// SIMATIC STEP 7 (V5.x) project TEMA 13 EJERCICIO 25
// CPU: CPU313 C-2 DP(1)
// station: P_ADR_BUS
// station: Hardware
// station: Equipo SIMATIC 300

DATA_BLOCK DB 1
VERSION : 0.1
  STRUCT
   M1 : BOOL ;
   M2 : BOOL ;
   M3 : BOOL ;
   M4 : BOOL ;
   M5 : BOOL ;
   M6 : BOOL ;
   M7 : BOOL ;
   M10 : BOOL ;
   M11 : BOOL ;
   M12 : BOOL ;
   M13 : BOOL ;
   M14 : BOOL ;
   M15 : BOOL ;
   M16 : BOOL ;
   M17 : BOOL ;
   M20 : BOOL ;
   M21 : BOOL ;
   M22 : BOOL ;
   M23 : BOOL ;
   M24 : BOOL ;
   M25 : BOOL ;
   M26 : BOOL ;
   M27 : BOOL ;
  END_STRUCT ;	
BEGIN
END_DATA_BLOCK

DATA_BLOCK DB 2
VERSION : 0.1
  STRUCT
   MARCA0 : BOOL ;
   MARCA1 : BOOL ;
   MARCA2 : BOOL ;
   MARCA3 : BOOL ;
   MARCA4 : BOOL ;
   MARCA5 : BOOL ;
   MARCA6 : BOOL ;
   MARCA7 : BOOL ;
   MARCA10 : BOOL ;
   MARCA11 : BOOL ;
   MARCA12 : BOOL ;
   MARCA13 : BOOL ;
   MARCA14 : BOOL ;
   MARCA15 : BOOL ;
   MARCA16 : BOOL ;
   MARCA17 : BOOL ;
  END_STRUCT ;	
BEGIN
END_DATA_BLOCK

DATA_BLOCK DB 3
VERSION : 0.1
  STRUCT
   MARCA0 : BOOL ;
   MARCA1 : BOOL ;
   MARCA2 : BOOL ;
   MARCA3 : BOOL ;
   MARCA4 : BOOL ;
   MARCA5 : BOOL ;
   MARCA6 : BOOL ;
   MARCA7 : BOOL ;
   MARCA10 : BOOL ;
   MARCA11 : BOOL ;
   MARCA12 : BOOL ;
   MARCA13 : BOOL ;
   MARCA14 : BOOL ;
   MARCA15 : BOOL ;
   MARCA16 : BOOL ;
   MARCA17 : BOOL ;
  END_STRUCT ;	
BEGIN
END_DATA_BLOCK

ORGANIZATION_BLOCK OB 1
TITLE = "Main Program Sweep (Cycle)"
//CLASIFICADOR AUTOMATICO DE CAJAS
VERSION : 0.1
VAR_TEMP
  OB1_EV_CLASS : BYTE ;	//Bits 0-3 = 1 (Coming event), Bits 4-7 = 1 (Event class 1)
  OB1_SCAN_1 : BYTE ;	//1 (Cold restart scan 1 of OB 1), 3 (Scan 2-n of OB 1)
  OB1_PRIORITY : BYTE ;	//Priority of OB Execution
  OB1_OB_NUMBR : BYTE ;	//1 (Organization block 1, OB1)
  OB1_RESERVED_1 : BYTE ;	//Reserved for system
  OB1_RESERVED_2 : BYTE ;	//Reserved for system
  OB1_PREV_CYCLE : INT ;	//Cycle time of previous OB1 scan (milliseconds)
  OB1_MIN_CYCLE : INT ;	//Minimum cycle time of OB1 (milliseconds)
  OB1_MAX_CYCLE : INT ;	//Maximum cycle time of OB1 (milliseconds)
  OB1_DATE_TIME : DATE_AND_TIME ;	//Date and time OB1 started
END_VAR
BEGIN
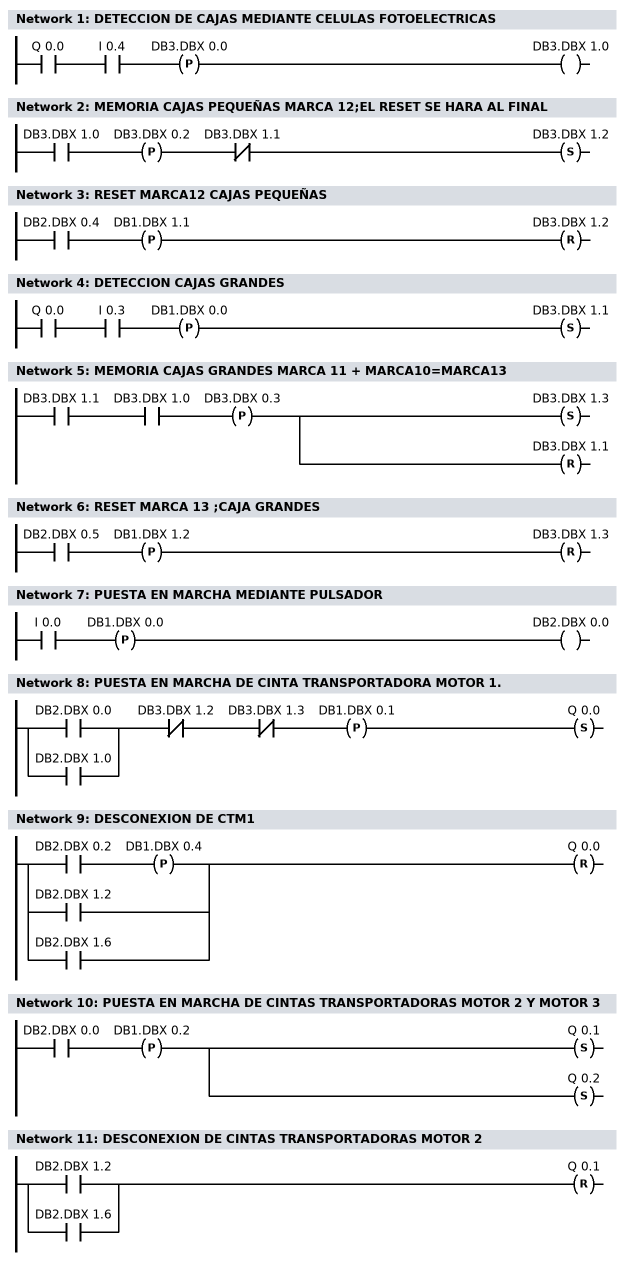
NETWORK
TITLE = DETECCION DE CAJAS MEDIANTE CELULAS FOTOELECTRICAS
//EXISTEN DOS TIPOS DE CAJAS PEQUEÑAS Y GRANDES.
//PARA RECONOCER LAS CAJAS PEQUEÑAS FCEL2 SE ACTIVARA YA QUE ESTA A LA ALTURA 
//OPORTUNA.
//PARA RECONOCER LAS CAJAS GRANDES SE TENDRA QUE ACTIVAR FCEL1 (NO PUEDE SER 
//ACTIVADO POR LAS CAJAS PEQUEÑAS POR QUE ESTA A LA ALTURA OPORTUNA)Y LUEGO FCEL2.
//ESTA INFORMACION SE TENDRA QUE GUARDAR EN UNA MEMORIA YA QUE EN CASO DE PARO,LA 
//MAQUINA UNA VEZ REANUDADA TENDRA QUE SEGUIR CON EL PROCESO CORRECTAMENTE.
//
//DETECCION CAJAS PEQUEÑAS
//
//
      A     Q 0.0;
      A     I 0.4;
      FP    DB3.DBX 0.0;
      =     DB3.DBX 1.0;
NETWORK
TITLE = MEMORIA CAJAS PEQUEÑAS MARCA 12;EL RESET SE HARA AL FINAL 
//COMO NECESITO QUE SE ACTIVE FCEL2 PARA REGISTRAR LA CAJAS GRANDES Y QUE NO ME 
//EJECUTE LA MEMORIA DE LAS PEQUEÑAS ,COLOCAREMOS OTRA MARCA AUXILIAR PARA QUE ME 
//PERMITA SUMAR LAS DOS SIN NECESIDAD DE CONFUNDIR A LA MAQUINA QUE SERA EN LA 
//CUAL INSERTE UN CONTACTO CERRADO PARA QUE SE HABRA UNA VEZ HALLA DETECTADO 
//FCEL1 Y ASI PODER UTILIZAR LA MARCA AUXILIAR.
      A     DB3.DBX 1.0;
      FP    DB3.DBX 0.2;
      AN    DB3.DBX 1.1;
      S     DB3.DBX 1.2;
NETWORK
TITLE = RESET MARCA12 CAJAS PEQUEÑAS
      A     DB2.DBX 0.4;
      FP    DB1.DBX 1.1;
      R     DB3.DBX 1.2;
NETWORK
TITLE = DETECCION CAJAS GRANDES
      A     Q 0.0;
      A     I 0.3;
      FP    DB1.DBX 0.0;
      S     DB3.DBX 1.1;
NETWORK
TITLE = MEMORIA CAJAS GRANDES MARCA 11 + MARCA10=MARCA13
//EL RESET DE LA MARCA SE HARA AL FINAL DEL PROCESO CUANDO YA NO SEA UTIL Y NOS 
//PERMITARA QUE LAS CELULAS FORTOELECTRICAS HAGAN SU FUNCION CORRECTAMENTE
      A     DB3.DBX 1.1;
      A     DB3.DBX 1.0;
      FP    DB3.DBX 0.3;
      S     DB3.DBX 1.3;
      R     DB3.DBX 1.1;
NETWORK
TITLE = RESET MARCA 13 ;CAJA GRANDES
      A     DB2.DBX 0.5;
      FP    DB1.DBX 1.2;
      R     DB3.DBX 1.3;
NETWORK
TITLE = PUESTA EN MARCHA MEDIANTE PULSADOR
//CUANDO PRESIONEMOS EL PULSADOR SE ACTIVARA EL PROCESO,ES DECIR,SE CONECTARAN 
//CTM1,CTM2,CTM3 Y LOS PISTONES ESTARAN PREPARADOS PARA CUANDO SEA NECESARIO
      A     I 0.0;
      FP    DB1.DBX 0.0;
      =     DB2.DBX 0.0;
NETWORK
TITLE = PUESTA EN MARCHA DE CINTA TRANSPORTADORA MOTOR 1.
//UN PULSO CONECTA CTM1 DE FORMA PERMANENTE
      A(;
      O     DB2.DBX 0.0;
      O     DB2.DBX 1.0;
      );
      AN    DB3.DBX 1.2;
      AN    DB3.DBX 1.3;
      FP    DB1.DBX 0.1;
      S     Q 0.0;
NETWORK
TITLE = DESCONEXION DE CTM1
//SE HARA EL RESET CUANDO CORRESPONDA:
//CUANDO LA CAJA PRESIONE EL F.C.FINAL LINEA.
//PARO.
//DESATIVACI0N.
      A     DB2.DBX 0.2;
      FP    DB1.DBX 0.4;
      O     DB2.DBX 1.2;
      O     DB2.DBX 1.6;
      R     Q 0.0;
NETWORK
TITLE = PUESTA EN MARCHA DE CINTAS TRANSPORTADORAS MOTOR 2 Y MOTOR 3 
//COMO ESTAS 2 CINTAS TRANSPORTADORAS FUNCIONAN  BAJO LAS MISMAS CONDIDICIONES 
//LOS 
//FACTORES QUE LAS CONECTAN Y DESCONECTAN SERAN LOS MISMOS.
      A     DB2.DBX 0.0;
      FP    DB1.DBX 0.2;
      S     Q 0.1;
      S     Q 0.2;
NETWORK
TITLE = DESCONEXION DE CINTAS TRANSPORTADORAS MOTOR 2  
//SE HARA EL RESET CUANDO CORRESPONDA:
//PARO.
//DESACTIVACION.
      O     DB2.DBX 1.2;
      O     DB2.DBX 1.6;
      R     Q 0.1;
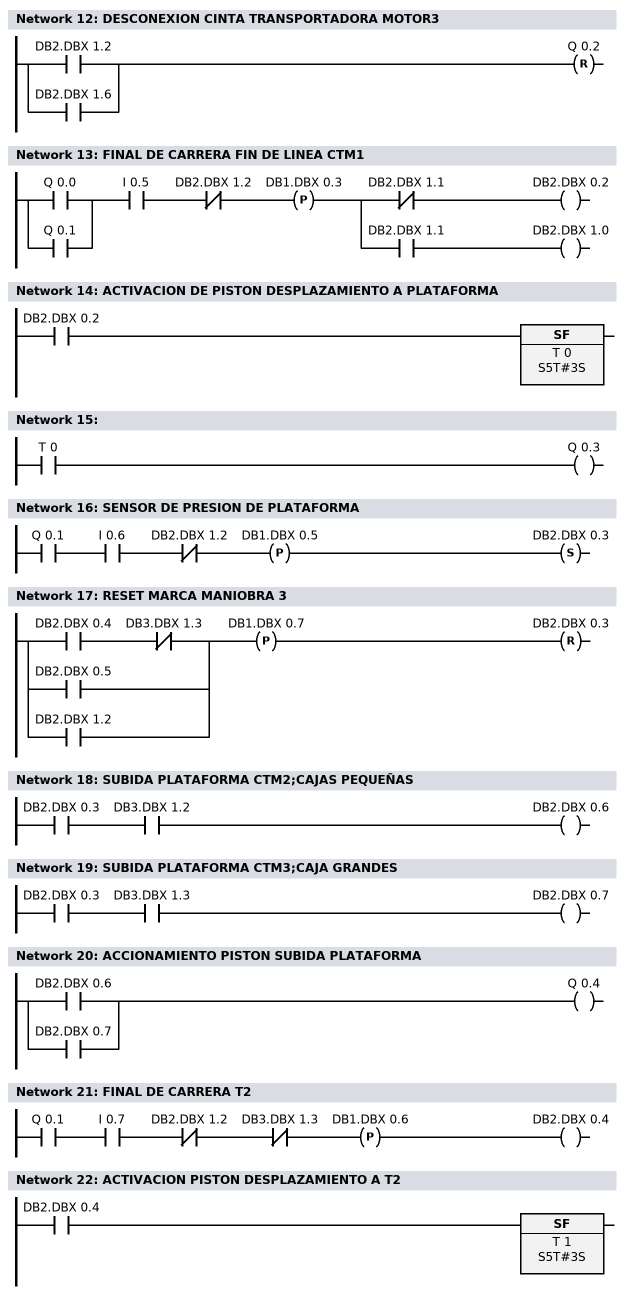
NETWORK
TITLE = DESCONEXION CINTA TRANSPORTADORA MOTOR3
//SE HARA EL RESET CUANDO CORRESPONDA:
//PARO.
//DESACTIVACION.
      O     DB2.DBX 1.2;
      O     DB2.DBX 1.6;
      R     Q 0.2;
NETWORK
TITLE = FINAL DE CARRERA FIN DE LINEA CTM1
//CUNADO UNA CAJA ACCIONE ESTE F.C. LA CTM1 SE PARARA Y ACTO SEGUIDO SE ACTIVARA 
//UN PISTON QUE DESPLAZARA LA CAJA SOBRE LA PLATAFORMA.
      A(;
      O     Q 0.0;
      O     Q 0.1;
      );
      A     I 0.5;
      AN    DB2.DBX 1.2;
      FP    DB1.DBX 0.3;
      =     L 20.0;
      A     L 20.0;
      AN    DB2.DBX 1.1;
      =     DB2.DBX 0.2;
      A     L 20.0;
      A     DB2.DBX 1.1;
      =     DB2.DBX 1.0;
NETWORK
TITLE = ACTIVACION DE PISTON DESPLAZAMIENTO A PLATAFORMA
//PARA SIMULAR EL ACCIONAMIENTO DE UN PISTON UTILIZO UN TEMPORIZADOR A LA 
//DESCONEXION QUE ALIMENTE UNA BOBINA(QUE ES EL PISTON) DURANTE 3 SEG.ES EL 
//TIEMPO 
//QUE TARDA EN DESPLAZARSE POR COMPLETO Y CUANDO SE APAGUE SE PRODUCIRA EL 
//RETORNO 
//POR RESORTE
      A     DB2.DBX 0.2;
      L     S5T#3S;
      SF    T 0;
NETWORK
TITLE =
      A     T 0;
      =     Q 0.3;
NETWORK
TITLE = SENSOR DE PRESION DE PLATAFORMA 
//UNA VEZ QUE EL SENSOR DE PRESION DETECTA UN PESO (EN ESTE CASO SERA CALIBRADO 
//PARA QUE CUALQUIERA DE LOS DOS TIPOS DE CAJAS LO ACTIVE) LA PLATAFORMA DEBERA 
//SUBIR A LA CINTA TRANSPORTADOA CORRESPODIENTE MEDIANTE UN PISTON 
      A     Q 0.1;
      A     I 0.6;
      AN    DB2.DBX 1.2;
      FP    DB1.DBX 0.5;
      S     DB2.DBX 0.3;
NETWORK
TITLE = RESET MARCA MANIOBRA 3
      A(;
      A     DB2.DBX 0.4;
      AN    DB3.DBX 1.3;
      O     DB2.DBX 0.5;
      O     DB2.DBX 1.2;
      );
      FP    DB1.DBX 0.7;
      R     DB2.DBX 0.3;
NETWORK
TITLE = SUBIDA PLATAFORMA CTM2;CAJAS PEQUEÑAS
//LA MARCA 12 ES LA QUE INDICA A LA PLATAFORMA DONDE TIENE QUE SUBIR Y SERA 
//INTERRUMPIDA POR SU FINAL DE CARRERA.CUANDO LAS MEMORIAS DE LAS CAJAS CAREZCAN 
//DE IMPORTANCIA SE HARA UN RESET
      A     DB2.DBX 0.3;
      A     DB3.DBX 1.2;
      =     DB2.DBX 0.6;
NETWORK
TITLE = SUBIDA PLATAFORMA CTM3;CAJA GRANDES
// LA MARCA 13 SE COMPORTA DE LA MISMA FORMA PERO SUBE HASTA CTM3
      A     DB2.DBX 0.3;
      A     DB3.DBX 1.3;
      =     DB2.DBX 0.7;
NETWORK
TITLE = ACCIONAMIENTO PISTON SUBIDA PLATAFORMA
      O     DB2.DBX 0.6;
      O     DB2.DBX 0.7;
      =     Q 0.4;
NETWORK
TITLE = FINAL DE CARRERA T2
//CUANDO SE ACCIONE SE PARARA LA SUBIDA DE LA PLATAFORMA E INICIARA SU RETROCESO 
//POR RESORTE,ACTIVARA EL PISTON DE DESPLAZAMIENTO A T2 Y HARA UN RESET DE LAS 
//MARCAS QUE YA NO SEAN UTILES PARA EL CORRECTO FUNCIONAMIENTO DEL PROCESO Y POR 
//LO TANTO ESTARAN PREPARADAS PARA LA SIGUIENTE SECUENCIA
      A     Q 0.1;
      A     I 0.7;
      AN    DB2.DBX 1.2;
      AN    DB3.DBX 1.3;
      FP    DB1.DBX 0.6;
      =     DB2.DBX 0.4;
NETWORK
TITLE = ACTIVACION PISTON DESPLAZAMIENTO A T2
//PARA SIMULAR EL PISTON UTILIZARE EL SISTEMA ANTERIOMENTE MENCIONADO
      A     DB2.DBX 0.4;
      L     S5T#3S;
      SF    T 1;
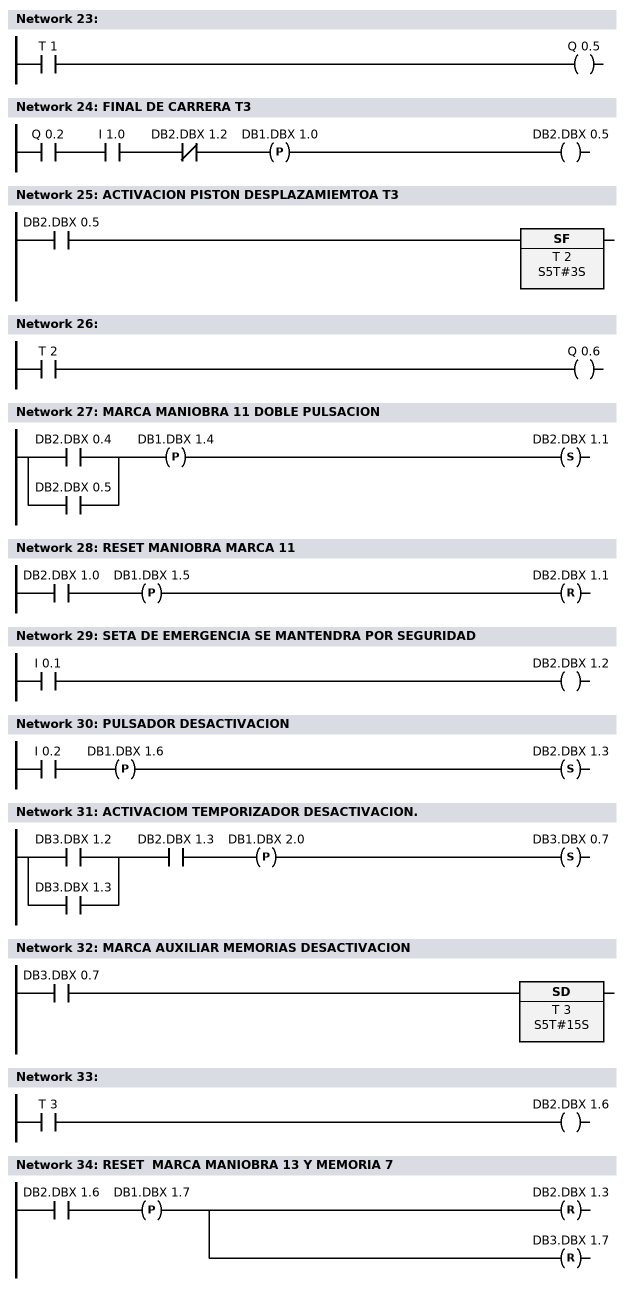
NETWORK
TITLE =
      A     T 1;
      =     Q 0.5;
NETWORK
TITLE = FINAL DE CARRERA T3
//EL SISTEMA SERA EL MISMO QUE EL ANTERIOMENTE CITADO
      A     Q 0.2;
      A     I 1.0;
      AN    DB2.DBX 1.2;
      FP    DB1.DBX 1.0;
      =     DB2.DBX 0.5;
NETWORK
TITLE = ACTIVACION PISTON DESPLAZAMIEMTOA T3
      A     DB2.DBX 0.5;
      L     S5T#3S;
      SF    T 2;
NETWORK
TITLE =
      A     T 2;
      =     Q 0.6;
NETWORK
TITLE = MARCA MANIOBRA 11 DOBLE PULSACION  
//CUANDO LA PLATAFORMA BAJE PRESIONARA OTRA VEZ EL F.C DE PLATAFORMA Y EN VEZ DE 
//PARAR CTM1 Y ACTIVAR PISTON DESPLAZAMIENTO SOLAMENTE ACTIVARA CTM1 Y LA 
//SIGUIENTE PULSACION PARARA CTM1 Y ACTIVARA PISTON. SE REPETIRA DE FORMA 
//INDEFINIDA.
      A(;
      O     DB2.DBX 0.4;
      O     DB2.DBX 0.5;
      );
      FP    DB1.DBX 1.4;
      S     DB2.DBX 1.1;
NETWORK
TITLE = RESET MANIOBRA MARCA 11
//SE HARA EL RESET CUANDO YA NO SEA NECESARIA,ES DECIR CUANDO ENTRE OTRA VEZ CTM1
      A     DB2.DBX 1.0;
      FP    DB1.DBX 1.5;
      R     DB2.DBX 1.1;
NETWORK
TITLE = SETA DE EMERGENCIA SE MANTENDRA POR SEGURIDAD
//AL PULSAR SE PARARA EL SISTEMA POR COMPLETO (LAS MEMORIAS DE MARCAS DE REGISTRO 
//DE CAJAS PERMANECERAN ACTIVAS PARA CUANDO SE ACTIVE EL SISTEMA DE NUEVO LA 
//MAQUINA SEPA DONDE SE ENCUENTRA Y ACTUE EN CONSECUENCIA) Y SE 
//CONDENARAN TODOS LOS FINALES DE CARRERA PARA EVITAR ACCIDENTES MIENTRAS SE 
//MANIPULE LA MAQUINA.
//MIENTRAS ESTE PRESIONADA LA SETA(RESET ALIMENTADO DE FORMA PERMANENTE) SERA 
//IMPOSIBLE HACER UN 
//SET EN LAS SALIDAS YA QUE PUEDE HABER RIESGO DE ACIONAMIENTO INVOLUNTARIO Y POR 
//LO TANTO UN FALLO FATAL.
//CONDICIONES DE PARO;
//PARO-LAS CINTAS ESTAN FUNCIONANDO,ES IRRELEVANTE.REINICIO NORMAL.
//PARO-FCEL1 DETECTA CAJA,ES IRRELEVANTE,LA MEMORIA PERMANECE REINICIO.NORMAL.
//PARO-FCEL2 DETECTA CAJA,ES IRRELEVANTE,LA MEMORIA PERMANECE REINICIO.NORMAL.
//PARO-CAJA PRESIONA F.C.F LINEA ,EL SIGUIENTE PASO SERIA DESCONECTAR CTM1 Y 
//ACTIVAR EL PISTON DE DESPLAZAMIENTO A PLATAFORMA UNA VEZ QUE HALLA DETECTADO 
//FCEL2 LA CAJA YA SE ENCUENTRA EN LA ZONA DE DESPLAZAMIENTO AL REINICIAR LA 
//MAQUINA ,EL F.C F LINEA ESTA PRESIONADO ASI QUE CTM1 NO FUNCIONA Y EL PISTON SE 
//DESPLAZA COLOCANDO LA CAJA EN LA PLATAFORMA.
//PARO-CAJA EN PLATAFORMA,EN ESTE CASO LAS MARCAS DE MEMORIA LAS QUE 
//INDIQUEN A LA MAQUINA DONDE SE ENCUENTRA Y DONDE DEBE DE IR(SI LA 
//PLATAFORMA ESTA SUBIENDO BAJARA A SU POSICION DE REPOSO).MARCHA CTM1 NO 
//FUNCIONA Y CTM2 Y CTM3 SI ,AL ESTAR PRESIONADO EL SENSOR DE PRESION LA 
//PLATAFORMA SUBIRA GOBERNADO POR LAS MARCAS DE MEMORIA DONDE CORRESPONDA.
      A     I 0.1;
      =     DB2.DBX 1.2;
NETWORK
TITLE = PULSADOR DESACTIVACION
//CON ESTE PULSADOR LO QUE CONSEGUINOS ES QUE EL SISTEMA DE FORMA INTELIGENTE 
//PARE 
//LA MAQUINA PERO NO AL INSTANTE ,EN EL CASO DE QUE HALLA INICIADO EL PROCESO(QUE 
//LAS CELULAS FOTOELECTRICAS HALLAN DETECTADO CAJA) DEJARA CONTINUAR HASTA 
//QUE TERMINE DE CLASIFICARLA Y NO PERMITIENDO QUE CIRCULE OTRA Y POR LO TANTO 
//ENTRA EN ESTADO DE REPOSO.CUANDO NO HALLA DETECTADO CAJA SE ACTIVARA LA 
//DESACTIVACION UNA VEZ ESTEN ACTIVAS LAS MARCAS DE MEMORIA 12 O 13.EL TIEMPO 
//ESTIMADO EN CLASIFICAR UNA CAJA DESDE QUE LAS CELULAS RECONOCEN CAJA HASTA QUE 
//LLEGAN A SU DESTINO ES DE 10 SEG.
//
      A     I 0.2;
      FP    DB1.DBX 1.6;
      S     DB2.DBX 1.3;
NETWORK
TITLE = ACTIVACIOM TEMPORIZADOR DESACTIVACION.
//PARA ACTUAR SOBRE ESTE TEMPORIZADOR UNA DE LAS MARCAS DE MEMORIA 12 O 13 TENDRAN
// 
//QUE ESTAR EN ON Y SI NO ES EL CASO ACTUARA CUANDO LO ESTE UNA DE LAS DOS.
      A(;
      O     DB3.DBX 1.2;
      O     DB3.DBX 1.3;
      );
      A     DB2.DBX 1.3;
      FP    DB1.DBX 2.0;
      S     DB3.DBX 0.7;
NETWORK
TITLE = MARCA AUXILIAR MEMORIAS DESACTIVACION
//ESTA MARCA NOS MANTENDRA EL TEMPORIZADOR , Y LA CONDICION PARA ACTIVARLA ES QUE 
//YA SE HALLAN ACTIVADO UNA DE LAS DOS Y LA MARCA DESACTIVACION.
      A     DB3.DBX 0.7;
      L     S5T#15S;
      SD    T 3;
NETWORK
TITLE =
      A     T 3;
      =     DB2.DBX 1.6;
NETWORK
TITLE = RESET  MARCA MANIOBRA 13 Y MEMORIA 7
      A     DB2.DBX 1.6;
      FP    DB1.DBX 1.7;
      R     DB2.DBX 1.3;
      R     DB3.DBX 1.7;
END_ORGANIZATION_BLOCK
